// TIA Portal project "piston_kol_hızı_hesaplama" (V18)

(* hardware
DEVICE "S7-1200 station_1"  S7-1200 Station
   slot 0: "Rack_0"  S7-1200 Rack  Rack  V1.0
   slot 1: "PLC_1"  CPU 1214C AC/DC/Rly  6ES7 214-1BG40-0XB0  V4.6
*)

// ===== PLC "PLC_1"  CPU 1214C AC/DC/Rly =====

VAR_GLOBAL   // PLC tag table "Default tag table"
   "piston dışarı" AT %I0.0 : Bool;
   "piston içeri" AT %I0.1 : Bool;
   "piston içeride" AT %I0.2 : Bool;
   "piston dışarıda" AT %I0.3 : Bool;
   "dış röle" AT %Q0.0 : Bool;
   "iç röle" AT %Q0.1 : Bool;
   "Tag_1" AT %M4.0 : Bool;
   "hız-mm/sn" AT %MD4 : DInt;
END_VAR

// folder: System blocks/Program resources

DATA_BLOCK "silindir zamanı"   // DB1
{ S7_Optimized_Access := 'TRUE' }
AUTHOR : Simatic
FAMILY : IEC
NAME : IEC_TMR
VERSION : 1.0
// stored: InstanceOfName IEC_TIMER
"IEC_TIMER"
BEGIN
END_DATA_BLOCK

// folder: (top level)

ORGANIZATION_BLOCK "Main"   // OB1, LAD, ProgramCycle
TITLE = "Main Program Sweep (Cycle)"
{ S7_Optimized_Access := 'TRUE' }
VERSION : 0.1
// UYGULAMA 32: Pnömatik bir silindirin piston koluna ait disari çikis hizi PLC ile
// hesaplanmak istenmektedir. Piston koluna ait hiz «mm/sn» cinsinden
// hesaplanacak ve kurs sonunda bir belle alaninda görülecektir. Silindir çift tarafli
// selenoid valf ile kumanda edilecektir.
// *Silindir kurs boyu 100 mm'dir.
// hız=yol/zaman
   VAR_INPUT
      Initial_Call : Bool;   // Initial call of this OB
      Remanence : Bool;   // =True, if remanent data are available
   END_VAR
   VAR_TEMP   // added for the SCL form of the ladder/FBD networks
      _w1 : Bool;
   END_VAR
BEGIN

REGION Network 1
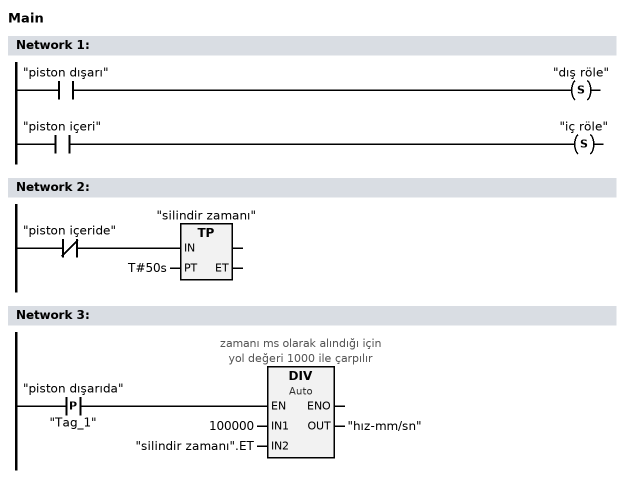
   RUNG wire#powerrail
      Contact( "piston dışarı" )
      S_Coil( "dış röle" )
   END_RUNG
   RUNG wire#powerrail
      Contact( "piston içeri" )
      S_Coil( "iç röle" )
   END_RUNG
   // the same network as SCL:
   IF "piston dışarı" THEN "dış röle" := TRUE; END_IF;
   IF "piston içeri" THEN "iç röle" := TRUE; END_IF;
END_REGION

REGION Network 2
   "silindir zamanı".TP(IN := NOT "piston içeride", PT := T#50s);
END_REGION

REGION Network 3
   RUNG wire#powerrail
      P_Contact(operand := "piston dışarıda", bit := "Tag_1")
      Div(in1 := 100000, in2 := "silindir zamanı".ET, out => "hız-mm/sn")   // zamanı ms olarak alındığı için yol değeri 1000 ile çarpılır
   END_RUNG
   // the same network as SCL:
   #_w1 := "piston dışarıda" AND NOT "Tag_1";   // rising edge of "piston dışarıda"
   "Tag_1" := "piston dışarıda";
   IF #_w1 THEN
       "hız-mm/sn" := 100000 / "silindir zamanı".ET;   // zamanı ms olarak alındığı için yol değeri 1000 ile çarpılır
   END_IF;
END_REGION
END_ORGANIZATION_BLOCK